FUNCTION_BLOCK FB_GenericUnit
VAR_IN_OUT
	bPumpOn: BOOL;
	
END_VAR
VAR_OUTPUT
END_VAR
VAR
END_VAR

M_Alarm();
M_Devices();

END_FUNCTION_BLOCK

(* stored: Version 1.1.0.1, ProductVersion 3.1.4024.12
   POU FB_GenericUnit: Id {95af2d81-bb8a-4668-a95a-43b2e7839b81}, SpecialFunc None *)
